RoboDK station: colur.rdk

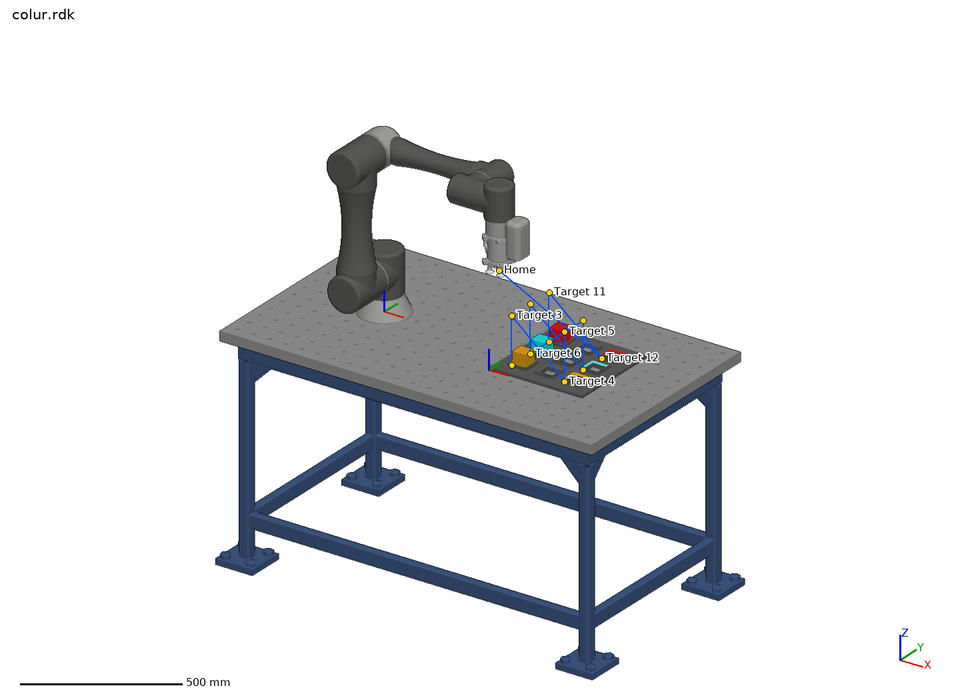
[picture v0: the station drawn from its stored meshes, robots at their saved joint values, targets as dots, program paths as lines]
Station colur (saved by RoboDK 5.9.2). Poses are relative to the parent item; angles as X-Y-Z fixed-axis rotations.
  - frame TM5-900 Base at (0, 0, 0) mm
    - robot TM5-900: 6 axes, payload 4 kg, reach 900 mm, repeatability 0.1 mm, weight 30 kg
        modified DH rows (alpha deg, a mm, theta deg, d mm): 0, 0, 0, 145.2; 90, 0, 90, 0; 0, 429, 0, 0; 0, 411, -90, 122.3; -90, 0, 0, 106.5; 90, 0, 180, 114.15
        joint limits [-360, -180, -155, -180, -180, -270] to [360, 180, 155, 180, 180, 270]; home [0, 0, 90, -90, 90, 0]; saved at [0, 0, 90, 0, 90, 0]
      - tool SMC ZXP7A01-ZP25C-X1 Vacuum Gripper, TCP at (0, 0, 125) mm, size 88 x 106.8 x 127.9 mm
  - object Table 1400x800x800mm at (0, 0, 0) mm, size 1420 x 820 x 800 mm, geometry from Table-1400x800x800mm.sld
  - frame Frame 2 at (500, -150, 0) mm
    - object Pallete  at (0, 0, 0) mm, size 350 x 350 x 20 mm, geometry from Pallete .step
    - target Home (Cartesian target) at (17.5, 27.7, 335.05) mm, rotated rx 180 ry 0 rz 90 deg; joints [0, 0, 90, 0, 90, 0] of TM5-900
    - target Target 3 (Cartesian target) at (50, 50, 180) mm, rotated rx 180 ry 0 rz 90 deg; joints [2.332, 7.612, 103.984, -21.596, 90, 2.332] of TM5-900
    - target Target 4 (Cartesian target) at (250, 50, 10) mm, rotated rx 180 ry 0 rz 90 deg; joints [1.707, 42.321, 78.934, -31.255, 90, 1.707] of TM5-900
    - target Target 5 (Cartesian target) at (250, 50, 180) mm, rotated rx 180 ry 0 rz 90 deg; joints [1.707, 33.646, 68.03, -11.677, 90, 1.707] of TM5-900
    - target Target 6 (Cartesian target) at (50, 150, 10) mm, rotated rx 180 ry 0 rz 90 deg; joints [12.848, 20.123, 116.526, -46.649, 90, 12.848] of TM5-900
    - target Target 7 (Cartesian target) at (50, 150, 180) mm, rotated rx 180 ry 0 rz 90 deg; joints [12.848, 6.426, 105.333, -21.758, 90, 12.848] of TM5-900
    - target Target 8 (Cartesian target) at (250, 150, 10) mm, rotated rx 180 ry 0 rz 90 deg; joints [9.385, 41.543, 80.349, -31.892, 90, 9.385] of TM5-900
    - target Target 9 (Cartesian target) at (250, 150, 180) mm, rotated rx 180 ry 0 rz 90 deg; joints [9.385, 32.703, 69.524, -12.227, 90, 9.385] of TM5-900
    - target Target 10 (Cartesian target) at (50, 250, 10) mm, rotated rx 180 ry 0 rz 90 deg; joints [22.942, 21.069, 115.076, -46.145, 90, 22.942] of TM5-900
    - target Target 11 (Cartesian target) at (50, 250, 180) mm, rotated rx 180 ry 0 rz 90 deg; joints [22.942, 7.612, 103.984, -21.596, 90, 22.942] of TM5-900
    - target Target 12 (Cartesian target) at (250, 250, 10) mm, rotated rx -180 ry 0 rz 90 deg; joints [16.897, 42.321, 78.934, -31.255, 90, 16.897] of TM5-900
    - target Target 2 (Cartesian target) at (50, 50, 10) mm, rotated rx 180 ry 0 rz 90 deg; joints [2.332, 21.069, 115.076, -46.145, 90, 2.332] of TM5-900
    - object yellow at (50, 50, 10) mm, size 50 x 50 x 50 mm, geometry from Cube-50mm.sld
    - object blue at (50, 150, 10) mm, size 50 x 50 x 50 mm, geometry from Cube-50mm.sld
    - object red at (50, 250, 10) mm, size 50 x 50 x 50 mm, geometry from Cube-50mm.sld
  - program Prog1 (1 instructions, listed below)
  - program Prog2 (20 instructions, listed below)
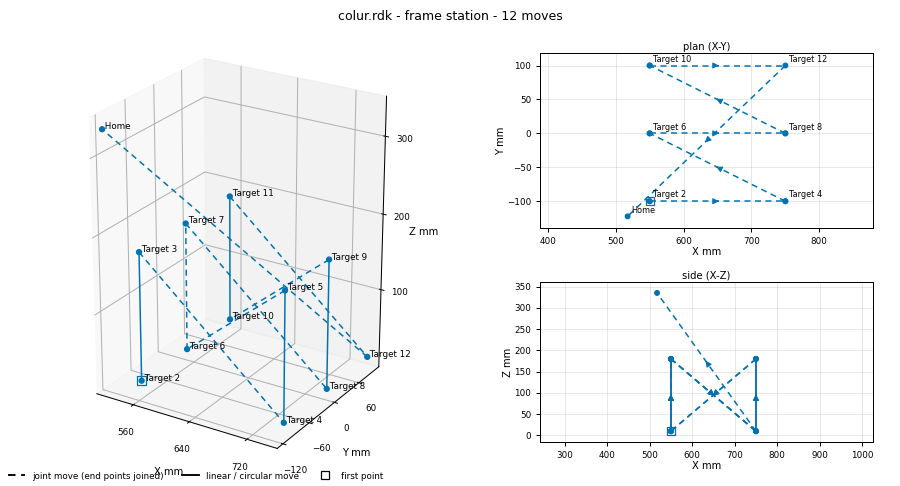
[picture p0: tool path of colur.rdk in frame station, 12 of 12 moves have a stored position in this frame; points joined in program order, loops and branches not executed]

--- program Prog1 (robot TM5-900) ---
  Replace objects

--- program Prog2 (robot TM5-900) ---
  Set Ref.: Frame 2
  Set Tool: SMC ZXP7A01-ZP25C-X1 Vacuum Gripper
  MoveJ (Target 2)
  Attach to SMC ZXP7A01-ZP25C-X1 Vacuum Gripper
  MoveL (Target 3)
  MoveJ (Target 4)
  Detach from SMC ZXP7A01-ZP25C-X1 Vacuum Gripper
  MoveL (Target 5)
  MoveJ (Target 6)
  Attach to SMC ZXP7A01-ZP25C-X1 Vacuum Gripper
  MoveJ (Target 7)
  MoveJ (Target 8)
  Detach from SMC ZXP7A01-ZP25C-X1 Vacuum Gripper
  MoveL (Target 9)
  MoveJ (Target 10)
  Attach to SMC ZXP7A01-ZP25C-X1 Vacuum Gripper
  MoveL (Target 11)
  MoveJ (Target 12)
  Detach from SMC ZXP7A01-ZP25C-X1 Vacuum Gripper
  MoveJ (Home)
